FUNCTION_BLOCK FBDelayCheck
VAR_INPUT
	in:INT;
	delaytime :TIME;  //T#0.2s
END_VAR

VAR_OUTPUT
	timeout_flag :BOOL;
	timeout_nums :INT;
END_VAR


VAR
	
	data1		:INT;
	fbRtrig 	:R_TRIG;
	fbTon 		:TON;
END_VAR


fbTon(IN:= (in = data1) ,PT:= delaytime);

fbRtrig(CLK:= fbTon.Q, Q=>timeout_flag);

IF timeout_flag THEN
	timeout_nums := timeout_nums+1;
END_IF

data1 :=in;

END_FUNCTION_BLOCK

(* stored: Version 1.1.0.1, ProductVersion 3.1.4022.18
   POU FBDelayCheck: Id {4c0e5754-e1f9-4158-a953-9d1af81ab7c1}, SpecialFunc None *)
